ABB RobotStudio station: InjectorSetUp.rsstnx

Station InjectorSetUp (saved by RobotStudio 24.4.11080.0)
Controller IRB4600_60_205_2
  mechanical unit ROB_1: IRB4600_60_205_C_01, 6 joints, base frame (0, 0, 0) mm
Layout (positions relative to the parent item):
  - BlackLeft [smart component, from Components\Attacher.rslib] at (-1000, 0, 0) mm
      properties: Parent=MoldGripper; Flange=0; Child=BlackLeft_Mold; Mount=false; Offset=[0 0 0]; Orientation=[0 0 0]
  - BlackRight_Mold [part] at (750, -1500, 1200) mm, rotated rx 90 ry 0 rz 90 deg, size 500 x 400 x 140 mm
  - BlackLeft_Mold [part] at (1000, -1000, 1200) mm, rotated rx 90 ry 0 rz -90 deg, size 505.4 x 403.2 x 145.2 mm
  - BlackLeft [smart component, from Components\LineSensor.rslib] at (-1000, 0, -91.46) mm
      properties: Start=[2 -0.98 1.39385]; End=[1.9 -0.98 1.39385]; Length=0.0999999999999999; Radius=0; Tag=(none); SensedPart=(none); SensedPoint=[0 0 0]
    - _sensorPart_ [part], size 100 x 0 x 0 mm
  - BlackLeft [smart component, from Components\Positioner.rslib] at (-1000, 0, 0) mm
      properties: Object=BlackLeft_Mold; Position=[1 -1 1.2]; Orientation=[1.5707963267949 0 -1.5707963267949]; Reference=Global; ReferenceObject=(none)
  - BlackLeft [smart component, from Components\Detacher.rslib] at (-1000, 0, 0) mm
      properties: Child=BlackLeft_Mold; KeepPosition=true
  - BaseMoldLeft [part] at (1800, 400, 1150) mm, size 504.9 x 145.6 x 402.9 mm
  - LetLeft [smart component, from Components\LineSensor.rslib] at (-1200, -37.49, 0) mm
      properties: Start=[2.985 0.38749 1.2]; End=[2.985 0.38749 1.4]; Length=0.2; Radius=0; Tag=(none); SensedPart=(none); SensedPoint=[0 0 0]
    - _sensorPart_ [part], size 0 x 0 x 200 mm
  - BlackRight [smart component, from Components\Positioner.rslib] at (-1000, 0, 0) mm
      properties: Object=BlackRight_Mold; Position=[0.75 -1.5 1.2]; Orientation=[1.5707963267949 0 1.5707963267949]; Reference=Global; ReferenceObject=(none)
  - BlackRight [smart component, from Components\Attacher.rslib] at (-1000, 0, 0) mm
      properties: Parent=MoldGripper; Flange=0; Child=BlackRight_Mold; Mount=false; Offset=[0 0 0]; Orientation=[0 0 0]
  - BlackRight [smart component, from Components\LineSensor.rslib] at (-1150, 0, -91.46) mm
      properties: Start=[2 -0.98 1.39385]; End=[1.9 -0.98 1.39385]; Length=0.1; Radius=0; Tag=(none); SensedPart=(none); SensedPoint=[0 0 0]
    - _sensorPart_ [part], size 100 x 0 x 0 mm
  - TakeRight [smart component, from Components\LineSensor.rslib] at (-1200, -800, -91.46) mm
      properties: Start=[2.985 0.75 1.39385]; End=[2.985 0.63252 1.39385]; Length=0.11748; Radius=0; Tag=(none); SensedPart=(none); SensedPoint=[0 0 0]
    - _sensorPart_ [part], size 0 x 117.5 x 0 mm
  - BlackRight [smart component, from Components\Detacher.rslib] at (-1000, 0, 0) mm
      properties: Child=BlackRight_Mold; KeepPosition=true
  - RedLeft_Mold [part] at (580, -1000, 1200) mm, rotated rx 90 ry 0 rz -90 deg, size 500 x 400 x 140 mm
  - RedRight_Mold [part] at (330, -1500, 1200) mm, rotated rx 90 ry 0 rz 90 deg, size 500 x 400 x 140 mm
  - BlueLeft_Mold [part] at (160, -1000, 1200) mm, rotated rx 90 ry 0 rz -90 deg, size 500 x 400 x 140 mm
  - BlueRight_Mold [part] at (-90, -1500, 1200) mm, rotated rx 90 ry 0 rz 90 deg, size 500 x 400 x 140 mm
  - RedLeft [smart component, from Components\Attacher.rslib] at (-1420, 0, 0) mm
      properties: Parent=MoldGripper; Flange=0; Child=RedLeft_Mold; Mount=false; Offset=[0 0 0]; Orientation=[0 0 0]
  - RedLeft [smart component, from Components\LineSensor.rslib] at (-1420, 0, -91.46) mm
      properties: Start=[2.42 -0.98 0.89385]; End=[2.32 -0.98 0.89385]; Length=0.0999999999999996; Radius=0; Tag=(none); SensedPart=(none); SensedPoint=[0 0 0]
    - _sensorPart_ [part], size 100 x 0 x 0 mm
  - RedLeft [smart component, from Components\Positioner.rslib] at (-1420, 0, 0) mm
      properties: Object=RedLeft_Mold; Position=[0.58 -1 1.2]; Orientation=[1.5707963267949 0 -1.5707963267949]; Reference=Global; ReferenceObject=(none)
  - RedLeft [smart component, from Components\Detacher.rslib] at (-1420, 0, 0) mm
      properties: Child=RedLeft_Mold; KeepPosition=true
  - RedRight [smart component, from Components\Positioner.rslib] at (-1420, 0, 0) mm
      properties: Object=RedRight_Mold; Position=[0.33 -1.5 1.2]; Orientation=[1.5707963267949 0 1.5707963267949]; Reference=Global; ReferenceObject=(none)
  - RedRight [smart component, from Components\Attacher.rslib] at (-1420, 0, 0) mm
      properties: Parent=MoldGripper; Flange=0; Child=RedRight_Mold; Mount=false; Offset=[0 0 0]; Orientation=[0 0 0]
  - RedRight [smart component, from Components\LineSensor.rslib] at (-1570, 0, -91.46) mm
      properties: Start=[2.42 -0.98 0.89385]; End=[2.32 -0.98 0.89385]; Length=0.1; Radius=0; Tag=(none); SensedPart=(none); SensedPoint=[0 0 0]
    - _sensorPart_ [part], size 100 x 0 x 0 mm
  - RedRight [smart component, from Components\Detacher.rslib] at (-1420, 0, 0) mm
      properties: Child=RedRight_Mold; KeepPosition=true
  - BlueLeft [smart component, from Components\Attacher.rslib] at (-1840, 0, 0) mm
      properties: Parent=MoldGripper; Flange=0; Child=BlueLeft_Mold; Mount=false; Offset=[0 0 0]; Orientation=[0 0 0]
  - BlueLeft [smart component, from Components\LineSensor.rslib] at (-1840, 0, -91.46) mm
      properties: Start=[2.84 -0.98 0.39385]; End=[2.74 -0.98 0.39385]; Length=0.0999999999999996; Radius=0; Tag=(none); SensedPart=(none); SensedPoint=[0 0 0]
    - _sensorPart_ [part], size 100 x 0 x 0 mm
  - BlueLeft [smart component, from Components\Positioner.rslib] at (-1840, 0, 0) mm
      properties: Object=BlueLeft_Mold; Position=[0.16 -1 1.2]; Orientation=[1.5707963267949 0 -1.5707963267949]; Reference=Global; ReferenceObject=(none)
  - BlueLeft [smart component, from Components\Detacher.rslib] at (-1840, 0, 0) mm
      properties: Child=BlueLeft_Mold; KeepPosition=true
  - BlueRight [smart component, from Components\Positioner.rslib] at (-1840, 0, 0) mm
      properties: Object=BlueRight_Mold; Position=[-0.09 -1.5 1.2]; Orientation=[1.5707963267949 0 1.5707963267949]; Reference=Global; ReferenceObject=(none)
  - BlueRight [smart component, from Components\Attacher.rslib] at (-1840, 0, 0) mm
      properties: Parent=MoldGripper; Flange=0; Child=BlueRight_Mold; Mount=false; Offset=[0 0 0]; Orientation=[0 0 0]
  - BlueRight [smart component, from Components\LineSensor.rslib] at (-1990, 0, -91.46) mm
      properties: Start=[2.84 -0.98 0.39385]; End=[2.74 -0.98 0.39385]; Length=0.0999999999999996; Radius=0; Tag=(none); SensedPart=(none); SensedPoint=[0 0 0]
    - _sensorPart_ [part], size 100 x 0 x 0 mm
  - BlueRight [smart component, from Components\Detacher.rslib] at (-1840, 0, 0) mm
      properties: Child=BlueRight_Mold; KeepPosition=true
  - InjectionMachine [part] at (1500, 1700, 0) mm, size 1314.8 x 3413.3 x 1819.5 mm
  - ClosePress [smart component, from Components\JointMover.rslib] at (-1000, 0, 0) mm
      properties: Mechanism=Press; Relative=false; Duration=1; J1=0.3
  - OpenPress [smart component, from Components\JointMover.rslib] at (-1000, 0, 0) mm
      properties: Mechanism=Press; Relative=false; Duration=1; J1=0
  - Press [mechanism] at (-1200, 0, 0) mm; joint values [0] (rad or m)
      links: Link1, Link2
  - LetRight [smart component, from Components\LineSensor.rslib] at (-1200, -800, 50) mm
      properties: Start=[3.51 0.67 1.34385]; End=[3.48 0.67 1.34385]; Length=0.0300000000000002; Radius=0; Tag=(none); SensedPart=(none); SensedPoint=[0 0 0]
    - _sensorPart_ [part], size 30 x 0 x 0 mm
  - PressBlackRight [smart component, from Components\Attacher.rslib] at (-1000, 0, 0) mm
      properties: Parent=Press; Flange=0; Child=BlackRight_Mold; Mount=false; Offset=[0 0 0]; Orientation=[0 0 0]
  - PressBlueRight [smart component, from Components\Attacher.rslib] at (-1000, 0, 0) mm
      properties: Parent=Press; Flange=0; Child=BlueRight_Mold; Mount=false; Offset=[0 0 0]; Orientation=[0 0 0]
  - PressRedRight [smart component, from Components\Attacher.rslib] at (-1000, 0, 0) mm
      properties: Parent=Press; Flange=0; Child=RedRight_Mold; Mount=false; Offset=[0 0 0]; Orientation=[0 0 0]
  - BlackRight [smart component, from Components\LogicGate.rslib]
      properties: Operator=AND; Delay=0
  - RedRight [smart component, from Components\LogicGate.rslib]
      properties: Operator=AND; Delay=0
  - BlueRight [smart component, from Components\LogicGate.rslib]
      properties: Operator=AND; Delay=0
  - BlackRight [smart component, from Components\VolumeSensor.rslib] at (-1000, 0, 0) mm
      properties: CornerPoint=[1.696 -1.51 1.19]; Orientation=[0 0 0]; Length=0.155; Width=0.522; Height=0.42; Tag=(none); PartialHit=false; SensedPart=BlackRight_Mold
    - _sensorPart_ [part], size 155 x 522 x 420 mm
  - BlackRight [smart component, from Components\LogicGate.rslib]
      properties: Operator=NOT; Delay=0
  - RedRight [smart component, from Components\VolumeSensor.rslib] at (-1000, 0, -500) mm
      properties: CornerPoint=[1.696 -1.51 1.19]; Orientation=[0 0 0]; Length=0.155; Width=0.522; Height=0.42; Tag=(none); PartialHit=false; SensedPart=(none)
    - _sensorPart_ [part], size 155 x 522 x 420 mm
  - BlueRight [smart component, from Components\VolumeSensor.rslib] at (-1000, 0, -1000) mm
      properties: CornerPoint=[1.696 -1.51 1.19]; Orientation=[0 0 0]; Length=0.155; Width=0.522; Height=0.42; Tag=(none); PartialHit=false; SensedPart=BlueRight_Mold
    - _sensorPart_ [part], size 155 x 522 x 420 mm
  - RedRight [smart component, from Components\LogicGate.rslib]
      properties: Operator=NOT; Delay=0
  - BlueRight [smart component, from Components\LogicGate.rslib]
      properties: Operator=NOT; Delay=0
  - BaseRight [smart component, from Components\VolumeSensor.rslib] at (-1200, 1000, 0) mm
      properties: CornerPoint=[2.998 -1.033 1.19]; Orientation=[0 0 -1.5707963267949]; Length=0.155; Width=0.522; Height=0.42; Tag=(none); PartialHit=false; SensedPart=(none)
    - _sensorPart_ [part], size 522 x 155 x 420 mm
  - BaseLeft [smart component, from Components\VolumeSensor.rslib] at (-1200, 1000, 0) mm
      properties: CornerPoint=[2.998 -0.595 1.19]; Orientation=[0 0 -1.5707963267949]; Length=0.155; Width=0.522; Height=0.42; Tag=(none); PartialHit=false; SensedPart=RedLeft_Mold
    - _sensorPart_ [part], size 522 x 155 x 420 mm
  - TakeRight [smart component, from Components\LogicGate.rslib]
      properties: Operator=AND; Delay=0
  - TakeRight [smart component, from Components\LogicGate.rslib]
      properties: Operator=NOT; Delay=0
  - BaseBlackRight [smart component, from Components\LogicGate.rslib]
      properties: Operator=AND; Delay=0
  - BaseBlackRight [smart component, from Components\Positioner.rslib] at (-1000, 0, 0) mm
      properties: Object=BlackRight_Mold; Position=[2.3 -0.13 1.2]; Orientation=[1.5707963267949 0 -3.14159265358979]; Reference=Global; ReferenceObject=(none)
  - BaseBlackLeft [smart component, from Components\Positioner.rslib] at (-1000, 0, 0) mm
      properties: Object=BlackLeft_Mold; Position=[1.8 0.35 1.2]; Orientation=[1.5707963267949 0 0]; Reference=Global; ReferenceObject=(none)
  - TakeLeft [smart component, from Components\LogicGate.rslib]
      properties: Operator=AND; Delay=0
  - BaseBlackLeft [smart component, from Components\LogicGate.rslib]
      properties: Operator=AND; Delay=0
  - TakeLeft [smart component, from Components\LineSensor.rslib] at (-1200, -420, -91.46) mm
      properties: Start=[2.985 0.7 1.39385]; End=[2.985 0.8 1.39385]; Length=0.1; Radius=0; Tag=(none); SensedPart=(none); SensedPoint=[0 0 0]
    - _sensorPart_ [part], size 0 x 100 x 0 mm
  - BlackLeft [smart component, from Components\VolumeSensor.rslib] at (-900, 0, 0) mm
      properties: CornerPoint=[1.8 -1.51 1.19]; Orientation=[0 0 0]; Length=0.155; Width=0.522; Height=0.42; Tag=(none); PartialHit=false; SensedPart=BlackLeft_Mold
    - _sensorPart_ [part], size 155 x 522 x 420 mm
  - RedLeft [smart component, from Components\VolumeSensor.rslib] at (-900, 0, -500) mm
      properties: CornerPoint=[1.8 -1.51 1.19]; Orientation=[0 0 0]; Length=0.155; Width=0.522; Height=0.42; Tag=(none); PartialHit=false; SensedPart=(none)
    - _sensorPart_ [part], size 155 x 522 x 420 mm
  - BlueLeft [smart component, from Components\VolumeSensor.rslib] at (-900, 0, -1000) mm
      properties: CornerPoint=[1.8 -1.51 1.19]; Orientation=[0 0 0]; Length=0.155; Width=0.522; Height=0.42; Tag=(none); PartialHit=false; SensedPart=BlueLeft_Mold
    - _sensorPart_ [part], size 155 x 522 x 420 mm
  - BlackLeft [smart component, from Components\LogicGate.rslib]
      properties: Operator=NOT; Delay=0
  - RedLeft [smart component, from Components\LogicGate.rslib]
      properties: Operator=NOT; Delay=0
  - BlueLeft [smart component, from Components\LogicGate.rslib]
      properties: Operator=NOT; Delay=0
  - BackBlackLeft [smart component, from Components\LineSensor.rslib] at (-1000, -521, 0) mm
      properties: Start=[2 -0.979 1.39385]; End=[1.9 -0.979 1.39385]; Length=0.0999999999999999; Radius=0; Tag=(none); SensedPart=BlackLeft_Mold; SensedPoint=[1 -1.5 1.39384997558594]
    - _sensorPart_ [part], size 100 x 0 x 0 mm
  - BackBlackRight [smart component, from Components\LineSensor.rslib] at (-1200, -521, 0) mm
      properties: Start=[2 -0.979 1.39385]; End=[1.9 -0.979 1.39385]; Length=0.0999999999999999; Radius=0; Tag=(none); SensedPart=BlackRight_Mold; SensedPoint=[0.788306640625 -1.5 1.39384997558594]
    - _sensorPart_ [part], size 100 x 0 x 0 mm
  - BackRedRight [smart component, from Components\LineSensor.rslib] at (-1200, -521, -500) mm
      properties: Start=[2 -0.979 1.39385]; End=[1.9 -0.979 1.39385]; Length=0.0999999999999999; Radius=0; Tag=(none); SensedPart=(none); SensedPoint=[0 0 0]
    - _sensorPart_ [part], size 100 x 0 x 0 mm
  - BackRedLeft [smart component, from Components\LineSensor.rslib] at (-1000, -521, -500) mm
      properties: Start=[2 -0.979 1.39385]; End=[1.9 -0.979 1.39385]; Length=0.0999999999999999; Radius=0; Tag=(none); SensedPart=(none); SensedPoint=[0 0 0]
    - _sensorPart_ [part], size 100 x 0 x 0 mm
  - BackBlueRight [smart component, from Components\LineSensor.rslib] at (-1200, -521, -1000) mm
      properties: Start=[2 -0.979 1.39385]; End=[1.9 -0.979 1.39385]; Length=0.0999999999999999; Radius=0; Tag=(none); SensedPart=BlueRight_Mold; SensedPoint=[0.788306640625 -1.5 0.393849975585937]
    - _sensorPart_ [part], size 100 x 0 x 0 mm
  - BackBlueLeft [smart component, from Components\LineSensor.rslib] at (-1000, -521, -1000) mm
      properties: Start=[2 -0.979 1.39385]; End=[1.9 -0.979 1.39385]; Length=0.0999999999999999; Radius=0; Tag=(none); SensedPart=BlueLeft_Mold; SensedPoint=[1 -1.5 0.393849975585937]
    - _sensorPart_ [part], size 100 x 0 x 0 mm
  - CloseTimer [smart component, from Components\Timer.rslib] at (-1000, 0, 0) mm
      properties: StartTime=1; Interval=0; Repeat=false; CurrentTime=10.992
  - OpenTimer [smart component, from Components\Timer.rslib]
      properties: StartTime=12; Interval=0; Repeat=false; CurrentTime=10.992
  - LogicSRLatch [smart component, from Components\LogicSRLatch.rslib]
  - BaseRedRight [smart component, from Components\LogicGate.rslib]
      properties: Operator=AND; Delay=0
  - BaseRedLeft [smart component, from Components\LogicGate.rslib]
      properties: Operator=AND; Delay=0
  - BaseBlueRight [smart component, from Components\LogicGate.rslib]
      properties: Operator=AND; Delay=0
  - BaseBlueLeft [smart component, from Components\LogicGate.rslib]
      properties: Operator=AND; Delay=0
  - ResetTimer [smart component, from Components\Timer.rslib]
      properties: StartTime=0.1; Interval=0; Repeat=false; CurrentTime=49.32
  - IRB4600_60_205_C_01 [mechanism, from %ABB.RobotStudio.Models.IRB4600%\IRB4600_60_205_C_G_01.rslib] at (0, 0, 0) mm; joint values [0.2755, -0.3031, 0.6212, 0.7351, -0.4177, -0.6907] (rad or m)
  - MoldGripper [mechanism] at (975, 237.5, 1220) mm, rotated rx 0 ry 90 rz 0 deg
      TCP MoldGripper at (0, -75, -20) mm, rotated rx 180 ry 0 rz -90 deg
      links: EndEffector
  - MoldsStore [part] at (675, -1600, 0) mm, size 400 x 600 x 1700 mm
  - Out1 [part] at (2210.58, -210, 320) mm, size 400 x 400 x 50 mm
  - FirstConveyor [part] at (1600, 190, 200) mm, size 2000 x 500 x 900 mm
  - MovementOut1 [smart component, from Components\MoveAlongCurve.rslib]
      properties: Object=Out1; WirePart=LineOut1; Speed=0.5; KeepOrientation=false; StartDistance=0; ResetPosition=true; StartPosition=[[1 0 0 0] [0 1 0 0] [0 0 1 0] [2.24 -0.21 0.32 1]]
  - MovementOut2 [smart component, from Components\MoveAlongCurve.rslib]
      properties: Object=Out2; WirePart=LineOut2; Speed=0.5; KeepOrientation=false; StartDistance=0; ResetPosition=false; StartPosition=[[1 0 0 0] [0 1 0 0] [0 0 1 0] [0 0 0 1]]
  - LineOut1 [part], size 240.6 x 0 x 0 mm
  - HideOut1 [smart component, from Components\Hide.rslib]
      properties: Object=Out1
  - HideOut2 [smart component, from Components\Hide.rslib]
      properties: Object=Out2
  - Out2 [part] at (2900.58, -211, 545) mm, rotated rx 0 ry -30 rz 0 deg, size 400 x 400 x 50 mm
  - ShowOut1 [smart component, from Components\Show.rslib]
      properties: Object=Out1
  - ShowOut2 [smart component, from Components\Show.rslib]
      properties: Object=Out2
  - LineOut2 [part], size 958.1 x 0 x 555.7 mm
  - PositionerOut1 [smart component, from Components\Positioner.rslib]
      properties: Object=Out1; Position=[2.210578 -0.21 0.32]; Orientation=[0 0 0]; Reference=Global; ReferenceObject=(none)
  - PositionerOut2 [smart component, from Components\Positioner.rslib]
      properties: Object=Out2; Position=[2.900578 -0.211 0.545]; Orientation=[0 -0.523598775598299 0]; Reference=Global; ReferenceObject=(none)
  - Blue1 [smart component, from Components\Highlighter.rslib]
      properties: Object=Out1; Color=[0 150 255]; Opacity=255
  - Blue2 [smart component, from Components\Highlighter.rslib]
      properties: Object=Out2; Color=[0 150 255]; Opacity=255
  - Red1 [smart component, from Components\Highlighter.rslib]
      properties: Object=Out1; Color=[255 0 0]; Opacity=255
  - Red2 [smart component, from Components\Highlighter.rslib]
      properties: Object=Out2; Color=[255 0 0]; Opacity=255
  - RedCount [smart component, from Components\Comparer.rslib]
      properties: ValueA=1; Operator===; ValueB=1
  - Counter_2 [smart component, from Components\Counter.rslib]
      properties: Count=1
  - BlueCount [smart component, from Components\Comparer.rslib]
      properties: ValueA=1; Operator===; ValueB=2
  - ResetCount [smart component, from Components\Comparer.rslib]
      properties: ValueA=1; Operator===; ValueB=3
  - OutSensor [smart component, from Components\LineSensor.rslib]
      properties: Start=[1.910578 0.19 0.38]; End=[1.910578 -0.21 0.38]; Length=0.4; Radius=0; Tag=(none); SensedPart=(none); SensedPoint=[0 0 0]
    - _sensorPart_ [part], size 0 x 400 x 0 mm
  - RealOut [part] at (2210.58, 80, 1550) mm, rotated rx -90 ry 0 rz 0 deg, size 400 x 400 x 50 mm
  - MovementRealOut [smart component, from Components\LinearMover2.rslib]
      properties: Object=RealOut; Direction=[0 0 -0.001]; Distance=0.8; Duration=0.404; Reference=Global; ReferenceObject=(none)
  - PositionerRealOut [smart component, from Components\Positioner.rslib]
      properties: Object=RealOut; Position=[2.210578 0.08 1.55]; Orientation=[-1.5707963267949 0 0]; Reference=Global; ReferenceObject=(none)
  - ShowRealOut [smart component, from Components\Show.rslib]
      properties: Object=RealOut
  - HideRealOut [smart component, from Components\Hide.rslib]
      properties: Object=RealOut
  - OpenPressAux [smart component, from Components\JointMover.rslib] at (-1000, 0, 0) mm
      properties: Mechanism=Press; Relative=false; Duration=1; J1=0
  - RedReal [smart component, from Components\Highlighter.rslib]
      properties: Object=RealOut; Color=[255 0 0]; Opacity=255
  - RealBlue [smart component, from Components\Highlighter.rslib]
      properties: Object=RealOut; Color=[0 150 255]; Opacity=255
  - Fence [graphiccomponentgroup]
    - Segment 1 [part], size 169.7 x 169.7 x 1400 mm
    - Segment 2 [part], size 169.7 x 1534.9 x 1400 mm
    - Segment 3 [part], size 1708.2 x 169.7 x 1400 mm
    - Segment 3 [part], size 1708.2 x 169.7 x 1400 mm
    - Segment 3 [part], size 1708.2 x 169.7 x 1400 mm
  - Fence_2 [graphiccomponentgroup]
    - Segment 1 [part], size 169.7 x 169.7 x 1400 mm
    - Segment 2 [part], size 120.3 x 1610.2 x 1400 mm
    - Segment 3 [part], size 1711.2 x 169.7 x 1400 mm
    - Segment 3 [part], size 1711.2 x 169.7 x 1400 mm
    - Segment 3 [part], size 1711.2 x 169.7 x 1400 mm
  - Fence_3 [graphiccomponentgroup]
    - Segment 1 [part], size 169.7 x 169.7 x 1400 mm
    - Segment 2 [part], size 316.7 x 1054.9 x 1400 mm
    - Segment 3 [part], size 169.7 x 1584.9 x 1400 mm
    - Segment 3 [part], size 169.7 x 1584.9 x 1400 mm
    - Segment 3 [part], size 169.7 x 1584.9 x 1400 mm
  - IRC5_Single-Cabinet [part, from %ABB.RobotStudio.Models.IRC5%\IRC5_Single-Cabinet.rslib] at (-4000, 800, 100) mm, rotated rx 90 ry 0 rz -90 deg
  - FlexPendant [part, from %ABB.RobotStudio.Models.IRC5%\FlexPendant.rslib] at (-3900, 980, 990) mm, rotated rx -27.17 ry 5.43 rz -119.59 deg
  - EnablingSwitch [part] at (-4070, 1000, 920) mm, rotated rx 0 ry 0 rz 180 deg, size 62.9 x 279 x 47.8 mm
  - Fence_4 [graphiccomponentgroup]
    - Segment 1 [part], size 169.7 x 169.7 x 1400 mm
    - Segment 2 [part], size 169.7 x 169.7 x 1400 mm
  - Pieza_1 [part], size 10 x 1000 x 10 mm
  - Pieza_31 [part] at (0, 0, -500) mm, size 10 x 1000 x 10 mm
  - Pieza_32 [part] at (0, 0, -1000) mm, size 10 x 1000 x 10 mm
Attachment: MoldGripper is attached to IRB4600_60_205_C_01 / Link6
Station signals: DI Digital1, DI Digital2
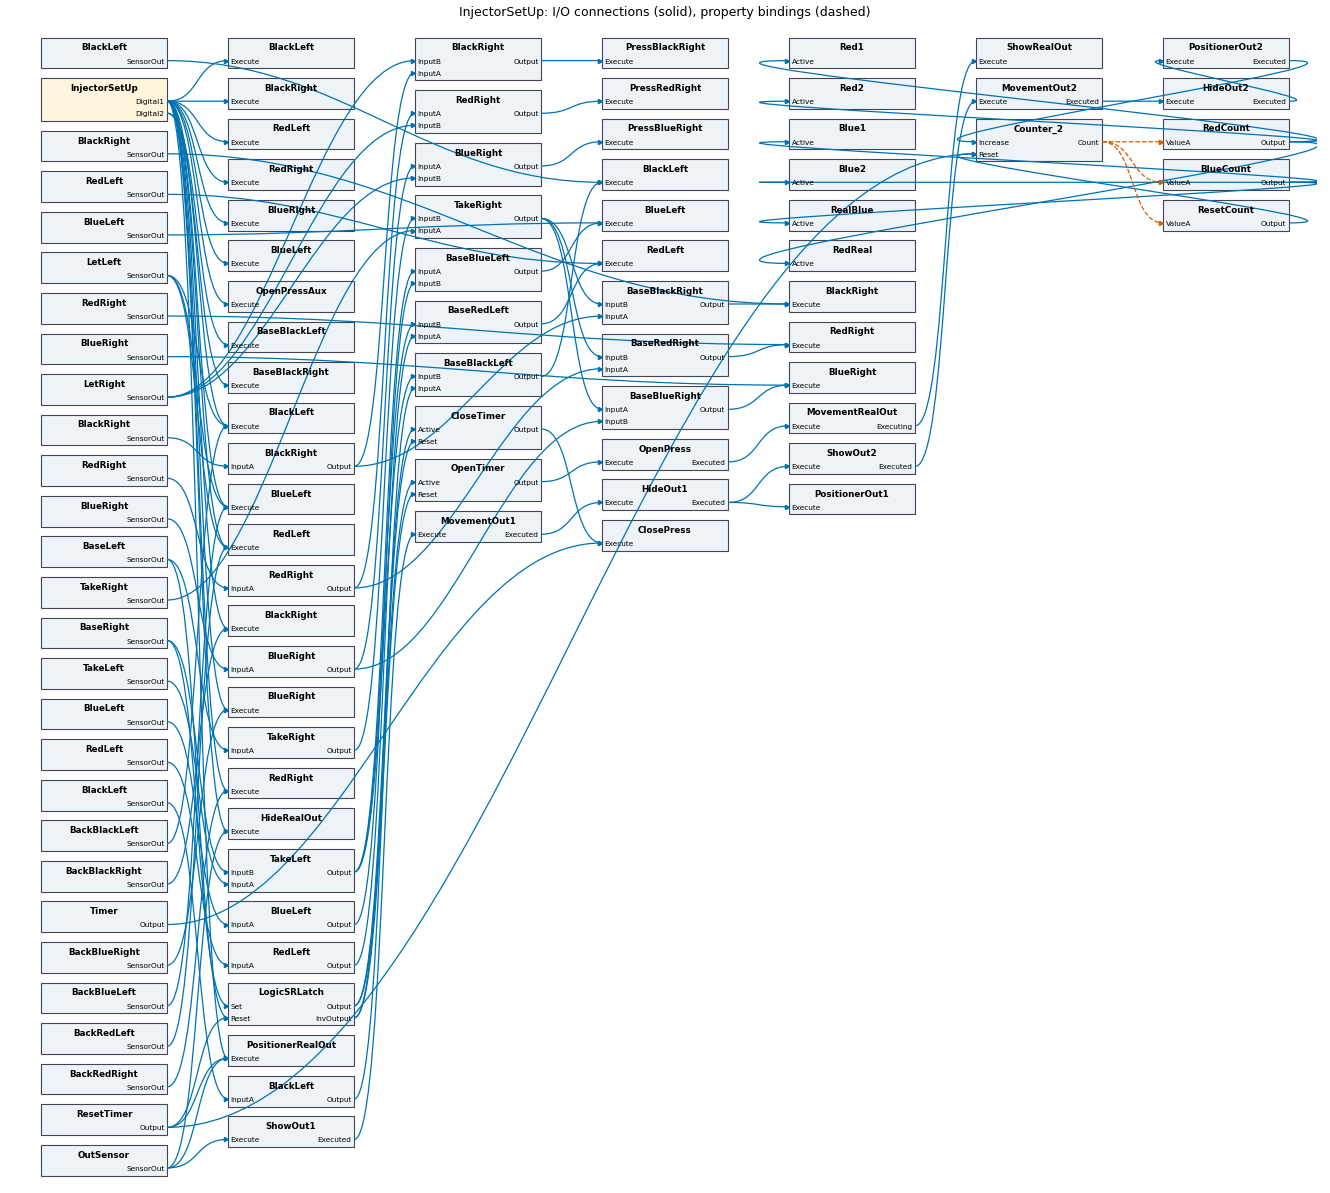
Station logic (signal -> signal, property => property):
  BlackLeft.SensorOut -> BlackLeft.Execute
  InjectorSetUp.Digital1 -> BlackLeft.Execute
  InjectorSetUp.Digital1 -> BlackLeft.Execute
  InjectorSetUp.Digital1 -> BlackRight.Execute
  BlackRight.SensorOut -> BlackRight.Execute
  InjectorSetUp.Digital1 -> BlackRight.Execute
  InjectorSetUp.Digital1 -> RedLeft.Execute
  InjectorSetUp.Digital1 -> BlueLeft.Execute
  InjectorSetUp.Digital1 -> RedRight.Execute
  InjectorSetUp.Digital1 -> BlueRight.Execute
  RedLeft.SensorOut -> RedLeft.Execute
  BlueLeft.SensorOut -> BlueLeft.Execute
  LetLeft.SensorOut -> BlackLeft.Execute
  LetLeft.SensorOut -> RedLeft.Execute
  LetLeft.SensorOut -> BlueLeft.Execute
  RedRight.SensorOut -> RedRight.Execute
  BlueRight.SensorOut -> BlueRight.Execute
  InjectorSetUp.Digital1 -> RedLeft.Execute
  InjectorSetUp.Digital1 -> RedRight.Execute
  InjectorSetUp.Digital1 -> BlueRight.Execute
  InjectorSetUp.Digital1 -> BlueLeft.Execute
  LetRight.SensorOut -> BlackRight.InputB
  BlackRight.SensorOut -> BlackRight.InputA
  BlackRight.Output -> BlackRight.InputA
  BlackRight.Output -> PressBlackRight.Execute
  RedRight.SensorOut -> RedRight.InputA
  RedRight.Output -> RedRight.InputA
  RedRight.Output -> PressRedRight.Execute
  BlueRight.SensorOut -> BlueRight.InputA
  BlueRight.Output -> BlueRight.InputA
  LetRight.SensorOut -> BlueRight.InputB
  LetRight.SensorOut -> RedRight.InputB
  BlueRight.Output -> PressBlueRight.Execute
  BaseLeft.SensorOut -> TakeRight.InputA
  TakeRight.Output -> TakeRight.InputB
  TakeRight.SensorOut -> TakeRight.InputA
  TakeRight.Output -> BaseBlackRight.InputB
  BaseBlackRight.Output -> BlackRight.Execute
  InjectorSetUp.Digital2 -> BaseBlackLeft.Execute
  InjectorSetUp.Digital2 -> BaseBlackRight.Execute
  BaseRight.SensorOut -> TakeLeft.InputB
  TakeLeft.SensorOut -> TakeLeft.InputA
  TakeLeft.Output -> BaseBlackLeft.InputB
  BlueLeft.SensorOut -> BlueLeft.InputA
  RedLeft.SensorOut -> RedLeft.InputA
  BlackLeft.SensorOut -> BlackLeft.InputA
  BlackLeft.Output -> BaseBlackLeft.InputA
  BaseBlackLeft.Output -> BlackLeft.Execute
  BlackRight.Output -> BaseBlackRight.InputA
  BackBlackLeft.SensorOut -> BlackLeft.Execute
  BackBlackRight.SensorOut -> BlackRight.Execute
  Timer.Output -> ClosePress.Execute
  CloseTimer.Output -> ClosePress.Execute
  OpenTimer.Output -> OpenPress.Execute
  BaseRight.SensorOut -> LogicSRLatch.Set
  LogicSRLatch.Output -> CloseTimer.Active
  LogicSRLatch.Output -> OpenTimer.Active
  BaseLeft.SensorOut -> LogicSRLatch.Reset
  LogicSRLatch.InvOutput -> OpenTimer.Reset
  LogicSRLatch.InvOutput -> CloseTimer.Reset
  BackBlueRight.SensorOut -> BlueRight.Execute
  BackBlueLeft.SensorOut -> BlueLeft.Execute
  BackRedLeft.SensorOut -> RedLeft.Execute
  BackRedRight.SensorOut -> RedRight.Execute
  TakeLeft.Output -> BaseRedLeft.InputB
  RedLeft.Output -> BaseRedLeft.InputA
  BaseRedLeft.Output -> RedLeft.Execute
  TakeRight.Output -> BaseRedRight.InputB
  RedRight.Output -> BaseRedRight.InputA
  BaseRedRight.Output -> RedRight.Execute
  TakeLeft.Output -> BaseBlueLeft.InputA
  BlueLeft.Output -> BaseBlueLeft.InputB
  BaseBlueLeft.Output -> BlueLeft.Execute
  TakeRight.Output -> BaseBlueRight.InputA
  BlueRight.Output -> BaseBlueRight.InputB
  BaseBlueRight.Output -> BlueRight.Execute
  ResetTimer.Output -> LogicSRLatch.Reset
  HideOut1.Executed -> ShowOut2.Execute
  ShowOut1.Executed -> MovementOut1.Execute
  ShowOut2.Executed -> MovementOut2.Execute
  MovementOut1.Executed -> HideOut1.Execute
  HideOut1.Executed -> PositionerOut1.Execute
  HideOut2.Executed -> PositionerOut2.Execute
  MovementOut2.Executed -> HideOut2.Execute
  PositionerOut2.Executed -> Counter_2.Increase
  RedCount.Output -> Red1.Active
  RedCount.Output -> Red2.Active
  BlueCount.Output -> Blue1.Active
  BlueCount.Output -> Blue2.Active
  ResetTimer.Output -> Counter_2.Reset
  ResetCount.Output -> Counter_2.Reset
  OutSensor.SensorOut -> PositionerRealOut.Execute
  OutSensor.SensorOut -> ShowOut1.Execute
  ResetTimer.Output -> PositionerRealOut.Execute
  OpenPress.Executed -> MovementRealOut.Execute
  InjectorSetUp.Digital1 -> PositionerRealOut.Execute
  OutSensor.SensorOut -> HideRealOut.Execute
  MovementRealOut.Executing -> ShowRealOut.Execute
  InjectorSetUp.Digital1 -> HideRealOut.Execute
  InjectorSetUp.Digital1 -> OpenPressAux.Execute
  BlueCount.Output -> RealBlue.Active
  RedCount.Output -> RedReal.Active
  Counter_2.Count => RedCount.ValueA
  Counter_2.Count => BlueCount.ValueA
  Counter_2.Count => ResetCount.ValueA
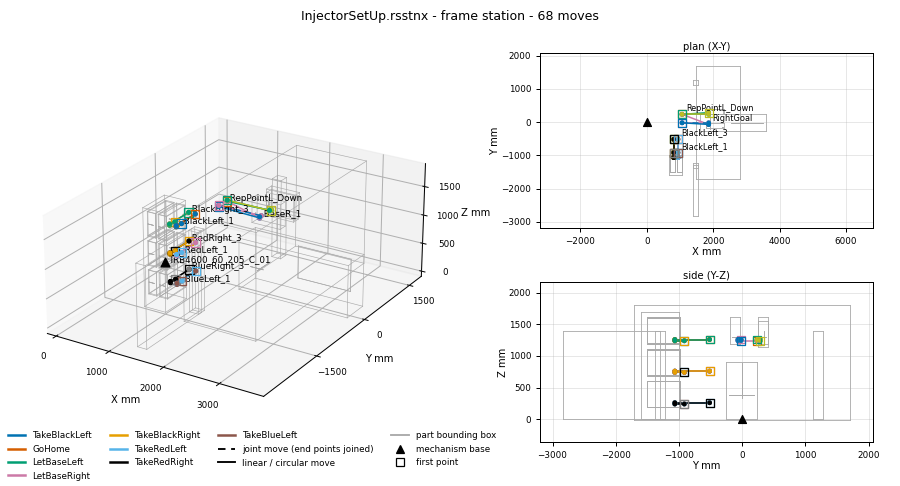
[picture p0: tool path of InjectorSetUp.rsstnx in frame station, 68 of 69 moves have a stored position in this frame; points joined in program order, loops and branches not executed]
Targets, tools, work objects and paths stored in the station, written as RAPID:
! task T_ROB1
MODULE CalibData
  PERS tooldata MoldGripper:=[TRUE,[[-20,0,90],[0.707106781,0,-0.707106781,0]],[56.229,[-0.255,0,9.024],[1,0,0,0],1.113132665,1.788384138,0.773824179]];
  TASK PERS wobjdata LeftBase:=[FALSE,TRUE,"",[[1800,400,1150],[1,0,0,0]],[[0,0,0],[1,0,0,0]]];
  TASK PERS wobjdata MoldsStore:=[FALSE,TRUE,"",[[910,-1000,1600],[0.707106781,0,0,-0.707106781]],[[0,0,0],[1,0,0,0]]];
  TASK PERS wobjdata RightBase:=[FALSE,TRUE,"",[[1800,-180,1150],[1,0,0,0]],[[0,0,0],[1,0,0,0]]];
ENDMODULE

! task T_ROB1
MODULE Module1
  CONST robtarget LeftGoal:=[[65,-112.5,110],[1,0,0,0],[0,0,-1,1],[9E+09,9E+09,9E+09,9E+09,9E+09,9E+09]];
  CONST robtarget BaseL_1:=[[65,-162.5,110],[1,0,0,0],[0,0,-1,1],[9E+09,9E+09,9E+09,9E+09,9E+09,9E+09]];
  CONST robtarget RepPointL_Up:=[[-735,-162.5,110],[1,0,0,0],[0,0,-1,1],[9E+09,9E+09,9E+09,9E+09,9E+09,9E+09]];
  CONST robtarget BaseL_2:=[[65,-112.5,90],[1,0,0,0],[0,0,-1,1],[9E+09,9E+09,9E+09,9E+09,9E+09,9E+09]];
  CONST robtarget RepPointL_Down:=[[-735,-162.5,90],[1,0,0,0],[0,0,-1,1],[9E+09,9E+09,9E+09,9E+09,9E+09,9E+09]];
  CONST robtarget BlackLeft_1:=[[-85,27.5,-360],[1,0,0,0],[-1,0,-1,1],[9E+09,9E+09,9E+09,9E+09,9E+09,9E+09]];
  CONST robtarget BlackLeft_2:=[[65,27.5,-360],[1,0,0,0],[-1,0,-1,1],[9E+09,9E+09,9E+09,9E+09,9E+09,9E+09]];
  CONST robtarget BlackLeft_Goal:=[[65,27.5,-340],[1,0,0,0],[-1,0,-1,1],[9E+09,9E+09,9E+09,9E+09,9E+09,9E+09]];
  CONST robtarget BlackRight_Goal:=[[65,-97.5,-340],[1,0,0,0],[-1,0,-1,1],[9E+09,9E+09,9E+09,9E+09,9E+09,9E+09]];
  CONST robtarget BlackRight_2:=[[65,-97.5,-360],[1,0,0,0],[-1,0,-1,1],[9E+09,9E+09,9E+09,9E+09,9E+09,9E+09]];
  CONST robtarget BlackRight_1:=[[-85,-97.5,-360],[1,0,0,0],[-1,0,-1,1],[9E+09,9E+09,9E+09,9E+09,9E+09,9E+09]];
  CONST robtarget BlackRight_3:=[[-485.000036812,-97.499955677,-340.00005254],[1,0.00000003,0.000000029,0.000000003],[-1,0,-1,1],[9E+09,9E+09,9E+09,9E+09,9E+09,9E+09]];
  CONST robtarget RedLeft_1:=[[-85,27.5,-860],[1,0,0,0],[-1,0,-1,1],[9E+09,9E+09,9E+09,9E+09,9E+09,9E+09]];
  CONST robtarget RedLeft_2:=[[65,27.5,-860],[1,0,0,0],[-1,0,-1,1],[9E+09,9E+09,9E+09,9E+09,9E+09,9E+09]];
  CONST robtarget RedLeft_Goal:=[[65,27.5,-840],[1,0,0,0],[-1,0,-1,1],[9E+09,9E+09,9E+09,9E+09,9E+09,9E+09]];
  CONST robtarget RedRight_1:=[[-85,-97.5,-860],[1,0,0,0],[-1,0,-1,1],[9E+09,9E+09,9E+09,9E+09,9E+09,9E+09]];
  CONST robtarget RedRight_2:=[[65,-97.5,-860],[1,0,0,0],[-1,0,-1,1],[9E+09,9E+09,9E+09,9E+09,9E+09,9E+09]];
  CONST robtarget RedRight_Goal:=[[65,-97.5,-840],[1,0,0,0],[-1,0,-1,1],[9E+09,9E+09,9E+09,9E+09,9E+09,9E+09]];
  CONST robtarget RedRight_3:=[[-485.000036812,-97.499955677,-840.00005254],[1,0.00000003,0.000000029,0.000000003],[-1,0,-1,1],[9E+09,9E+09,9E+09,9E+09,9E+09,9E+09]];
  CONST robtarget BlueLeft_1:=[[-85,27.5,-1360],[1,0,0,0],[-1,0,-1,1],[9E+09,9E+09,9E+09,9E+09,9E+09,9E+09]];
  CONST robtarget BlueLeft_2:=[[65,27.5,-1360],[1,0,0,0],[-1,0,-1,1],[9E+09,9E+09,9E+09,9E+09,9E+09,9E+09]];
  CONST robtarget BlueLeft_Goal:=[[65,27.5,-1340],[1,0,0,0],[-1,0,-1,1],[9E+09,9E+09,9E+09,9E+09,9E+09,9E+09]];
  CONST robtarget BlueRight_1:=[[-85,-97.5,-1360],[1,0,0,0],[-1,0,-1,1],[9E+09,9E+09,9E+09,9E+09,9E+09,9E+09]];
  CONST robtarget BlueRight_2:=[[65,-97.5,-1360],[1,0,0,0],[-1,0,-1,1],[9E+09,9E+09,9E+09,9E+09,9E+09,9E+09]];
  CONST robtarget BlueRight_Goal:=[[65,-97.5,-1340],[1,0,0,0],[-1,0,-1,1],[9E+09,9E+09,9E+09,9E+09,9E+09,9E+09]];
  CONST robtarget BlueRight_3:=[[-485.000036812,-97.499955677,-1340.00005254],[1,0.00000003,0.000000029,0.000000003],[-1,0,-1,1],[9E+09,9E+09,9E+09,9E+09,9E+09,9E+09]];
  CONST robtarget BlackLeft_3:=[[-485,27.5,-340],[1,0,0,0],[-1,0,-1,1],[9E+09,9E+09,9E+09,9E+09,9E+09,9E+09]];
  CONST robtarget RedLeft_3:=[[-485,27.5,-840],[1,0,0,0],[-1,0,-1,1],[9E+09,9E+09,9E+09,9E+09,9E+09,9E+09]];
  CONST robtarget BlueLeft_3:=[[-485,27.5,-1340],[1,0,0,0],[-1,0,-1,1],[9E+09,9E+09,9E+09,9E+09,9E+09,9E+09]];
  CONST robtarget RightGoal:=[[65,112.5,110],[1,0,0,0],[-1,-1,0,1],[9E+09,9E+09,9E+09,9E+09,9E+09,9E+09]];
  CONST robtarget BaseR_1:=[[65,162.5,110],[1,0,0,0],[-1,-1,0,1],[9E+09,9E+09,9E+09,9E+09,9E+09,9E+09]];
  CONST robtarget RepPointR_Up:=[[-734.999864723,162.499998844,109.999989577],[1,0,-0.000000004,0],[-1,-1,0,1],[9E+09,9E+09,9E+09,9E+09,9E+09,9E+09]];
  CONST robtarget BaseR_2:=[[65,112.5,90],[1,0,0,0],[-1,-1,0,1],[9E+09,9E+09,9E+09,9E+09,9E+09,9E+09]];
  CONST robtarget RepPointR_Down:=[[-735,162.5,90],[1,0,0,0],[-1,-1,0,1],[9E+09,9E+09,9E+09,9E+09,9E+09,9E+09]];
  CONST jointtarget Rest:=[[0,-60,60,0,30,0],[9E+09,9E+09,9E+09,9E+09,9E+09,9E+09]];
  PROC GoRest()
    MoveAbsJ Rest,robotSpeed,z200,MoldGripper\WObj:=wobj0;
  ENDPROC
  PROC TakeBlackLeft()
    MoveJ BlackLeft_1,robotSpeed,fine,MoldGripper\WObj:=MoldsStore;
    MoveL BlackLeft_2,robotSpeed,fine,MoldGripper\WObj:=MoldsStore;
    MoveL BlackLeft_Goal,robotSpeed,fine,MoldGripper\WObj:=MoldsStore;
    MoveL BlackLeft_3,robotSpeed,z100,MoldGripper\WObj:=MoldsStore;
  ENDPROC
  PROC main()
    velocity;
    GoRest;
    CycleBlack;
    CycleRed;
    CycleBlue;
    GoHome;
  ENDPROC
  PROC GoHome()
    MoveJ RepPointL_Down,robotSpeed,z200,MoldGripper\WObj:=LeftBase;
  ENDPROC
  PROC LetBaseLeft()
    MoveL RepPointL_Up,robotSpeed,fine,MoldGripper\WObj:=LeftBase;
    MoveL BaseL_1,robotSpeed,fine,MoldGripper\WObj:=LeftBase;
    MoveL LeftGoal,robotSpeed,fine,MoldGripper\WObj:=LeftBase;
    MoveL BaseL_2,robotSpeed,fine,MoldGripper\WObj:=LeftBase;
    MoveL RepPointL_Down,robotSpeed,fine,MoldGripper\WObj:=LeftBase;
  ENDPROC
  PROC LetBaseRight()
    MoveL RepPointR_Up,robotSpeed,fine,MoldGripper\WObj:=RightBase;
    MoveL BaseR_1,robotSpeed,fine,MoldGripper\WObj:=RightBase;
    MoveL RightGoal,robotSpeed,fine,MoldGripper\WObj:=RightBase;
    MoveL BaseR_2,robotSpeed,fine,MoldGripper\WObj:=RightBase;
    MoveL RepPointL_Down,robotSpeed,fine,MoldGripper\WObj:=LeftBase;
  ENDPROC
  PROC TakeBlackRight()
    MoveJ BlackRight_1,robotSpeed,fine,MoldGripper\WObj:=MoldsStore;
    MoveL BlackRight_2,robotSpeed,fine,MoldGripper\WObj:=MoldsStore;
    MoveL BlackRight_Goal,robotSpeed,fine,MoldGripper\WObj:=MoldsStore;
    MoveL BlackRight_3,robotSpeed,z100,MoldGripper\WObj:=MoldsStore;
  ENDPROC
  PROC TakeRedLeft()
    MoveJ RedLeft_1,robotSpeed,fine,MoldGripper\WObj:=MoldsStore;
    MoveL RedLeft_2,robotSpeed,fine,MoldGripper\WObj:=MoldsStore;
    MoveL RedLeft_Goal,robotSpeed,fine,MoldGripper\WObj:=MoldsStore;
    MoveL RedLeft_3,robotSpeed,z100,MoldGripper\WObj:=MoldsStore;
  ENDPROC
  PROC TakeRedRight()
    MoveJ RedRight_1,robotSpeed,fine,MoldGripper\WObj:=MoldsStore;
    MoveL RedRight_2,robotSpeed,fine,MoldGripper\WObj:=MoldsStore;
    MoveL RedRight_Goal,robotSpeed,fine,MoldGripper\WObj:=MoldsStore;
    MoveL RedRight_3,robotSpeed,z100,MoldGripper\WObj:=MoldsStore;
  ENDPROC
  PROC TakeBlueLeft()
    MoveJ BlueLeft_1,robotSpeed,fine,MoldGripper\WObj:=MoldsStore;
    MoveL BlueLeft_2,robotSpeed,fine,MoldGripper\WObj:=MoldsStore;
    MoveL BlueLeft_Goal,robotSpeed,fine,MoldGripper\WObj:=MoldsStore;
    MoveL BlueLeft_3,robotSpeed,z100,MoldGripper\WObj:=MoldsStore;
  ENDPROC
  PROC TakeBlueRight()
    MoveJ BlueRight_1,robotSpeed,fine,MoldGripper\WObj:=MoldsStore;
    MoveL BlueRight_2,robotSpeed,fine,MoldGripper\WObj:=MoldsStore;
    MoveL BlueRight_Goal,robotSpeed,fine,MoldGripper\WObj:=MoldsStore;
    MoveL BlueRight_3,robotSpeed,z100,MoldGripper\WObj:=MoldsStore;
  ENDPROC
  PROC TakeBaseLeft()
    MoveL BaseL_2,robotSpeed,fine,MoldGripper\WObj:=LeftBase;
    MoveL LeftGoal,robotSpeed,fine,MoldGripper\WObj:=LeftBase;
    MoveL BaseL_1,robotSpeed,fine,MoldGripper\WObj:=LeftBase;
    MoveL RepPointL_Up,robotSpeed,fine,MoldGripper\WObj:=LeftBase;
  ENDPROC
  PROC TakeBaseRight()
    MoveJ RepPointR_Down,robotSpeed,fine,MoldGripper\WObj:=RightBase;
    MoveL BaseR_2,robotSpeed,fine,MoldGripper\WObj:=RightBase;
    MoveL RightGoal,robotSpeed,fine,MoldGripper\WObj:=RightBase;
    MoveL BaseR_1,robotSpeed,fine,MoldGripper\WObj:=RightBase;
    MoveJ RepPointR_Up,robotSpeed,fine,MoldGripper\WObj:=RightBase;
  ENDPROC
  PROC LetBlackLeft()
    TakeBlackLeft;
    LetBaseLeft;
  ENDPROC
  PROC LetBlackRight()
    TakeBlackRight;
    LetBaseRight;
  ENDPROC
  PROC LetRedLeft()
    TakeRedLeft;
    LetBaseLeft;
  ENDPROC
  PROC LetRedRight()
    TakeRedRight;
    LetBaseRight;
  ENDPROC
  PROC LetBlueLeft()
    TakeBlueLeft;
    LetBaseLeft;
  ENDPROC
  PROC LetBlueRight()
    TakeBlueRight;
    LetBaseRight;
  ENDPROC
  PROC ReturnBlackLeft()
    MoveJ BlackLeft_3,robotSpeed,z100,MoldGripper\WObj:=MoldsStore;
    MoveL BlackLeft_Goal,robotSpeed,fine,MoldGripper\WObj:=MoldsStore;
    MoveL BlackLeft_2,robotSpeed,fine,MoldGripper\WObj:=MoldsStore;
    MoveL BlackLeft_1,robotSpeed,fine,MoldGripper\WObj:=MoldsStore;
  ENDPROC
  PROC ReturnBlackRight()
    MoveJ BlackRight_3,robotSpeed,z100,MoldGripper\WObj:=MoldsStore;
    MoveL BlackRight_Goal,robotSpeed,fine,MoldGripper\WObj:=MoldsStore;
    MoveL BlackRight_2,robotSpeed,fine,MoldGripper\WObj:=MoldsStore;
    MoveL BlackRight_1,robotSpeed,fine,MoldGripper\WObj:=MoldsStore;
  ENDPROC
  PROC ReturnRedLeft()
    MoveJ RedLeft_3,robotSpeed,z100,MoldGripper\WObj:=MoldsStore;
    MoveL RedLeft_Goal,robotSpeed,fine,MoldGripper\WObj:=MoldsStore;
    MoveL RedLeft_2,robotSpeed,fine,MoldGripper\WObj:=MoldsStore;
    MoveL RedLeft_1,robotSpeed,fine,MoldGripper\WObj:=MoldsStore;
  ENDPROC
  PROC ReturnRedRight()
    MoveJ RedRight_3,robotSpeed,z100,MoldGripper\WObj:=MoldsStore;
    MoveL RedRight_Goal,robotSpeed,fine,MoldGripper\WObj:=MoldsStore;
    MoveL RedRight_2,robotSpeed,fine,MoldGripper\WObj:=MoldsStore;
    MoveL RedRight_1,robotSpeed,fine,MoldGripper\WObj:=MoldsStore;
  ENDPROC
  PROC ReturnBlueLeft()
    MoveJ BlueLeft_3,robotSpeed,z100,MoldGripper\WObj:=MoldsStore;
    MoveL BlueLeft_Goal,robotSpeed,fine,MoldGripper\WObj:=MoldsStore;
    MoveL BlueLeft_2,robotSpeed,fine,MoldGripper\WObj:=MoldsStore;
    MoveL BlueLeft_1,robotSpeed,fine,MoldGripper\WObj:=MoldsStore;
  ENDPROC
  PROC ReturnBlueRight()
    MoveJ BlueRight_3,robotSpeed,z100,MoldGripper\WObj:=MoldsStore;
    MoveL BlueRight_Goal,robotSpeed,fine,MoldGripper\WObj:=MoldsStore;
    MoveL BlueRight_2,robotSpeed,fine,MoldGripper\WObj:=MoldsStore;
    MoveL BlueRight_1,robotSpeed,fine,MoldGripper\WObj:=MoldsStore;
  ENDPROC
  PROC BackBlackLeft()
    TakeBaseLeft;
    ReturnBlackLeft;
  ENDPROC
  PROC BackBlackRight()
    TakeBaseRight;
    ReturnBlackRight;
  ENDPROC
  PROC BackRedLeft()
    TakeBaseLeft;
    ReturnRedLeft;
  ENDPROC
  PROC BackRedRight()
    TakeBaseRight;
    ReturnRedRight;
  ENDPROC
  PROC BackBlueLeft()
    TakeBaseLeft;
    ReturnBlueLeft;
  ENDPROC
  PROC BackBlueRight()
    TakeBaseRight;
    ReturnBlueRight;
  ENDPROC
  PROC CycleBlack()
    LetBlackLeft;
    LetBlackRight;
    WaitTime 23;
    BackBlackLeft;
    BackBlackRight;
  ENDPROC
  PROC CycleRed()
    LetRedLeft;
    LetRedRight;
    WaitTime 23;
    BackRedLeft;
    BackRedRight;
  ENDPROC
  PROC CycleBlue()
    LetBlueLeft;
    LetBlueRight;
    WaitTime 23;
    BackBlueLeft;
    BackBlueRight;
  ENDPROC
  PROC velocity()
  ENDPROC
ENDMODULE

! task T_ROB1
MODULE Module1
  PROC TakeBlackLeft()
  ENDPROC
  PROC main()
    GoHome;
    CycleBlack;
    CycleRed;
    CycleBlue;
    GoHome;
  ENDPROC
  PROC GoHome()
  ENDPROC
  PROC LetBaseLeft()
  ENDPROC
  PROC LetBaseRight()
  ENDPROC
  PROC TakeBlackRight()
  ENDPROC
  PROC TakeRedLeft()
  ENDPROC
  PROC TakeRedRight()
  ENDPROC
  PROC TakeBlueLeft()
  ENDPROC
  PROC TakeBlueRight()
  ENDPROC
  PROC TakeBaseLeft()
  ENDPROC
  PROC TakeBaseRight()
  ENDPROC
  PROC LetBlackLeft()
    TakeBlackLeft;
    LetBaseLeft;
  ENDPROC
  PROC LetBlackRight()
    TakeBlackRight;
    LetBaseRight;
  ENDPROC
  PROC LetRedLeft()
    TakeRedLeft;
    LetBaseLeft;
  ENDPROC
  PROC LetRedRight()
    TakeRedRight;
    LetBaseRight;
  ENDPROC
  PROC LetBlueLeft()
    TakeBlueLeft;
    LetBaseLeft;
  ENDPROC
  PROC LetBlueRight()
    TakeBlueRight;
    LetBaseRight;
  ENDPROC
  PROC ReturnBlackLeft()
  ENDPROC
  PROC ReturnBlackRight()
  ENDPROC
  PROC ReturnRedLeft()
  ENDPROC
  PROC ReturnRedRight()
  ENDPROC
  PROC ReturnBlueLeft()
  ENDPROC
  PROC ReturnBlueRight()
  ENDPROC
  PROC BackBlackLeft()
    TakeBaseLeft;
    ReturnBlackLeft;
  ENDPROC
  PROC BackBlackRight()
    TakeBaseRight;
    ReturnBlackRight;
  ENDPROC
  PROC BackRedLeft()
    TakeBaseLeft;
    ReturnRedLeft;
  ENDPROC
  PROC BackRedRight()
    TakeBaseRight;
    ReturnRedRight;
  ENDPROC
  PROC BackBlueLeft()
    TakeBaseLeft;
    ReturnBlueLeft;
  ENDPROC
  PROC BackBlueRight()
    TakeBaseRight;
    ReturnBlueRight;
  ENDPROC
  PROC CycleBlack()
    LetBlackLeft;
    LetBlackRight;
    WaitTime 23;
    BackBlackLeft;
    BackBlackRight;
  ENDPROC
  PROC CycleRed()
    LetRedLeft;
    LetRedRight;
    WaitTime 23;
    BackRedLeft;
    BackRedRight;
  ENDPROC
  PROC CycleBlue()
    LetBlueLeft;
    LetBlueRight;
    WaitTime 23;
    BackBlueLeft;
    BackBlueRight;
  ENDPROC
ENDMODULE

